// TIA Portal project "Project2" (V16)

(* hardware
DEVICE "S7300/ET200M station_1"  S7-300 station
   slot 0: "Rail_0"  Rail  6ES7 390-1***0-0AA0
   slot 2: "PLC_1"  CPU 317-2 PN/DP  6ES7 317-2EK14-0AB0  V3.2
      slot 2: "PROFINET interface_1"  PN-IO
         slot 1: "Port_1"  Port
         slot 2: "Port_2"  Port
   slot 4: "DI 16x24VDC_1"  DI16 x 24VDC, interrupt  6ES7 321-7BH01-0AB0
   slot 5: "DO 16x24VDC/0.5A_1"  DO16 x 24VDC / 0.5A  6ES7 322-1BH01-0AA0
*)

// ===== PLC "PLC_1"  CPU 317-2 PN/DP =====

VAR_GLOBAL   // PLC tag table "Default tag table"
   "dButton1" AT %I0.0 : Bool;
   "dButton2" AT %I0.1 : Bool;
   "dButton3" AT %I0.2 : Bool;
   "mTemp" AT %M0.0 : Bool;
   "doLamp1" AT %Q0.0 : Bool;
   "doLamp2" AT %Q0.1 : Bool;
   "doLamp3" AT %Q0.2 : Bool;
END_VAR

ORGANIZATION_BLOCK "Main"   // OB1, LAD
TITLE = "Main Program Sweep (Cycle)"
{ S7_Optimized_Access := 'FALSE' }
VERSION : 0.1
   VAR_TEMP
      OB1_EV_CLASS : Byte;   // Bits 0-3 = 1 (Coming event), Bits 4-7 = 1 (Event class 1)
      OB1_SCAN_1 : Byte;   // 1 (Cold restart scan 1 of OB 1), 3 (Scan 2-n of OB 1)
      OB1_PRIORITY : Byte;   // Priority of OB Execution
      OB1_OB_NUMBR : Byte;   // 1 (Organization block 1, OB1)
      OB1_RESERVED_1 : Byte;   // Reserved for system
      OB1_RESERVED_2 : Byte;   // Reserved for system
      OB1_PREV_CYCLE : Int;   // Cycle time of previous OB1 scan (milliseconds)
      OB1_MIN_CYCLE : Int;   // Minimum cycle time of OB1 (milliseconds)
      OB1_MAX_CYCLE : Int;   // Maximum cycle time of OB1 (milliseconds)
      OB1_DATE_TIME : Date_And_Time;   // Date and time OB1 started
   END_VAR
BEGIN

REGION Network 1
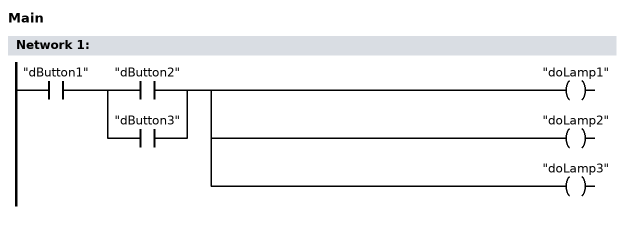
   RUNG wire#powerrail
      Contact( "dButton1" )
      wire#w1
      Contact( "dButton2" )
      wire#w2
      Coil( "doLamp1" )
   END_RUNG
   RUNG wire#w1
      Contact( "dButton3" )
   END_RUNG wire#w2
   RUNG wire#w2
      Coil( "doLamp2" )
   END_RUNG
   RUNG wire#w2
      Coil( "doLamp3" )
   END_RUNG
   // the same network as SCL:
   "doLamp1" := "dButton1" AND ("dButton2" OR "dButton3");
   "doLamp2" := "doLamp1";
   "doLamp3" := "doLamp1";
END_REGION
END_ORGANIZATION_BLOCK